{attribute 'GeneratedUsingTerminal: EL1502-0000-0001'}
{attribute addProperty BoxType "EL1502-0000-0001"}
{attribute addProperty Id "EtcSlaveTerminalBaseCNT_InputsAT %I*CNT_Inputs_147BF88E12CNT_OutputsAT %Q*CNT_Outputs_EB14A6758WcStateAT %I*WcState_9091E0EB2InfoDataAT %I*InfoData_32EB74EA10"}
{attribute addProperty CRC "1613473371"}
{attribute addProperty Size "32"}
TYPE EL1502_602BA65B EXTENDS EtcSlaveTerminalBase :
STRUCT
	{attribute addProperty Name "CNT_Inputs"}
	CNT_Inputs : CNT_Inputs_147BF88E;
	{attribute addProperty Name "CNT_Outputs"}
	CNT_Outputs : CNT_Outputs_EB14A675;
	{attribute addProperty Name "WcState"}
	WcState : WcState_9091E0EB;
	{attribute addProperty Name "InfoData"}
	InfoData : InfoData_32EB74EA;
END_STRUCT
END_TYPE

(* stored: Version 1.2.0.0, ProductVersion 3.1.4024.9
   DUT EL1502_602BA65B: Id {5876ceb9-119a-4199-9f5d-411a0e71f73a} *)
